(* Logix 5000 project; controller NSH_PLC1 vendor 1 type 14 code 167 rev 32.11; software revision 32.02; part 5 of 12 *)
(* tags used below, declared in another part *)
   H10 : Motor;   // Auger
   H14A : Motor;   // Shr. Roll
   H14B : Motor;   // Shr. Roll
   H15A : Motor;   // Aspirator
   H15B : Motor;   // Aspirator
   H20A : Motor;   // Shr. Roll
   H20B : Motor;   // Shr. Roll
   H20C : Motor;   // Vib.
   H21A : Motor;   // Aspirator
   H21B : Motor;   // Aspirator
   H25 : Motor;   // Ele.
   H26 : Motor;   // Auger
   H27 : Motor;   // Auger
   H28A : Motor;   // HC Vib.
   H28B : Motor;   // Hard Crkr.
   H28C : Motor;   // S.Roll
   H28D : Motor;   // Shr.Roll.
   H29A : Motor;   // Aspirator
   H29B : Motor;   // Aspirator
   H30 : Motor;   // Auger
   H31 : Motor;   // Roll Fdr.
   H32A : Motor;   // HS Cracker
   H32B : Motor;   // Hard Crkr.
   H32C : Motor;   // Shr.Roll.
   H32D : Motor;   // Shr.Roll.
   H33A : Motor;   // Aspirator
   H33B : Motor;   // Aspirator
   H34A : Motor;   // HC Vib.
   H34B : Motor;   // Hard Crkr.
   H34C : Motor;   // S.Roll
   H34D : Motor;   // Shr.Roll.
   H35A : Motor;   // Aspirator
   H35B : Motor;   // Aspirator
   H36 : Motor;   // BMM
   H37A : Motor;   // Aspirator
   H37B : Motor;   // Aspirator
   H38A : Motor;   // Aspirator
   H38B : Motor;   // Aspirator
   H39 : Motor;   // Ele.
   H40 : Motor;   // Auger
   H41 : Motor;   // Auger
   H42A : Motor;   // HC Vib.
   H42B : Motor;   // Hard Crkr.
   H42C : Motor;   // S.Roll
   H42D : Motor;   // Shr.Roll.
   H44A : Motor;   // HC Vib.
   H44B : Motor;   // Hard Crkr.
   H44C : Motor;   // S.Roll
   H44D : Motor;   // Shr.Roll.
   H45A : Motor;   // Aspirator
   H45B : Motor;   // Aspirator
   H46 : Motor;   // BMM
   H47A : Motor;   // Aspirator
   H47B : Motor;   // Aspirator
   H48A : Motor;   // Aspirator
   H48B : Motor;   // Aspirator
(* HullerSheller, continued *)

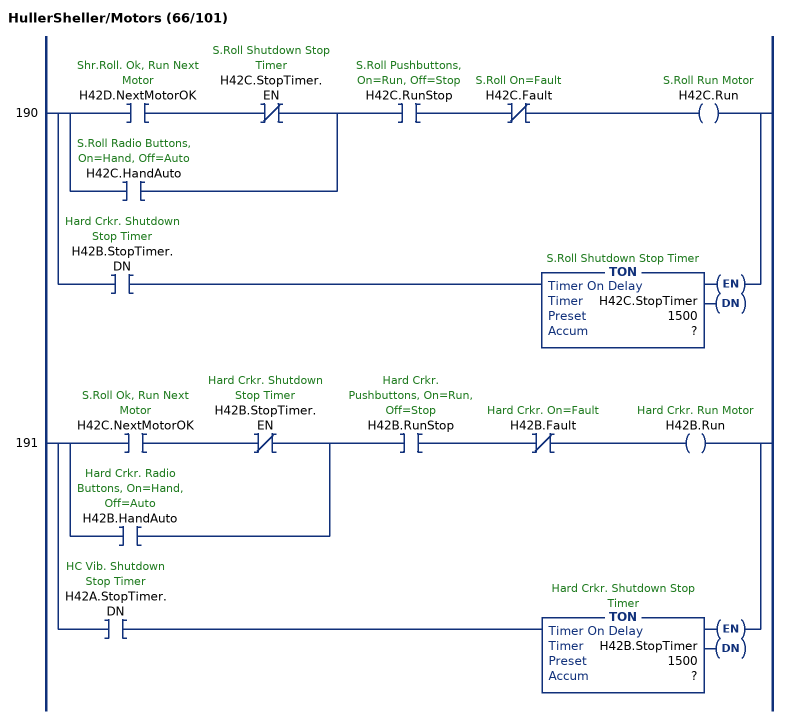
   [picture p90: HullerSheller/Motors rungs 190-191]
   190: [[XIC(H42D.NextMotorOK) XIO(H42C.StopTimer.EN) ,XIC(H42C.HandAuto) ] XIC(H42C.RunStop) XIO(H42C.Fault) OTE(H42C.Run) ,XIC(H42B.StopTimer.DN) TON(H42C.StopTimer,?,?) ];
   191: [[XIC(H42C.NextMotorOK) XIO(H42B.StopTimer.EN) ,XIC(H42B.HandAuto) ] XIC(H42B.RunStop) XIO(H42B.Fault) OTE(H42B.Run) ,XIC(H42A.StopTimer.DN) TON(H42B.StopTimer,?,?) ];
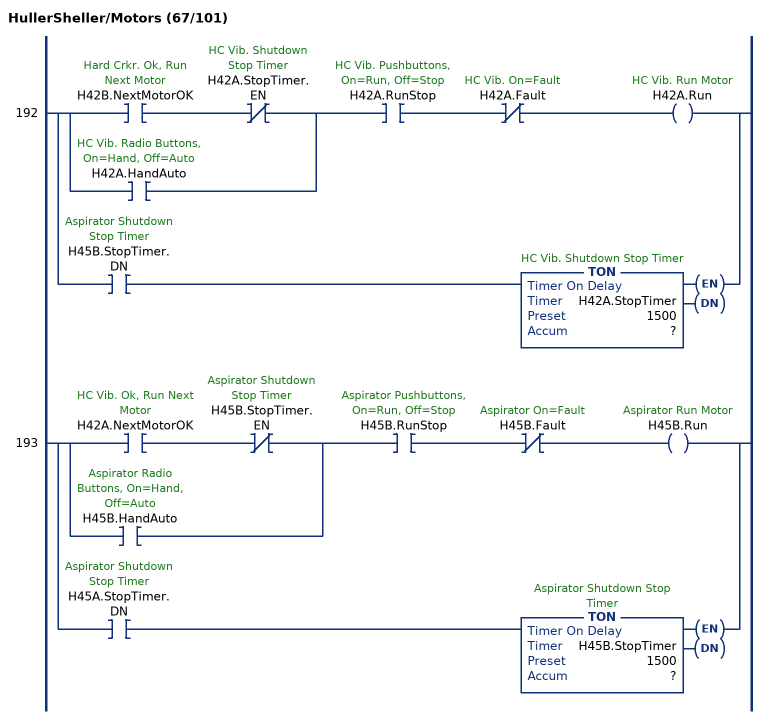
   192: [[XIC(H42B.NextMotorOK) XIO(H42A.StopTimer.EN) ,XIC(H42A.HandAuto) ] XIC(H42A.RunStop) XIO(H42A.Fault) OTE(H42A.Run) ,XIC(H45B.StopTimer.DN) TON(H42A.StopTimer,?,?) ];
   193: [[XIC(H42A.NextMotorOK) XIO(H45B.StopTimer.EN) ,XIC(H45B.HandAuto) ] XIC(H45B.RunStop) XIO(H45B.Fault) OTE(H45B.Run) ,XIC(H45A.StopTimer.DN) TON(H45B.StopTimer,?,?) ];
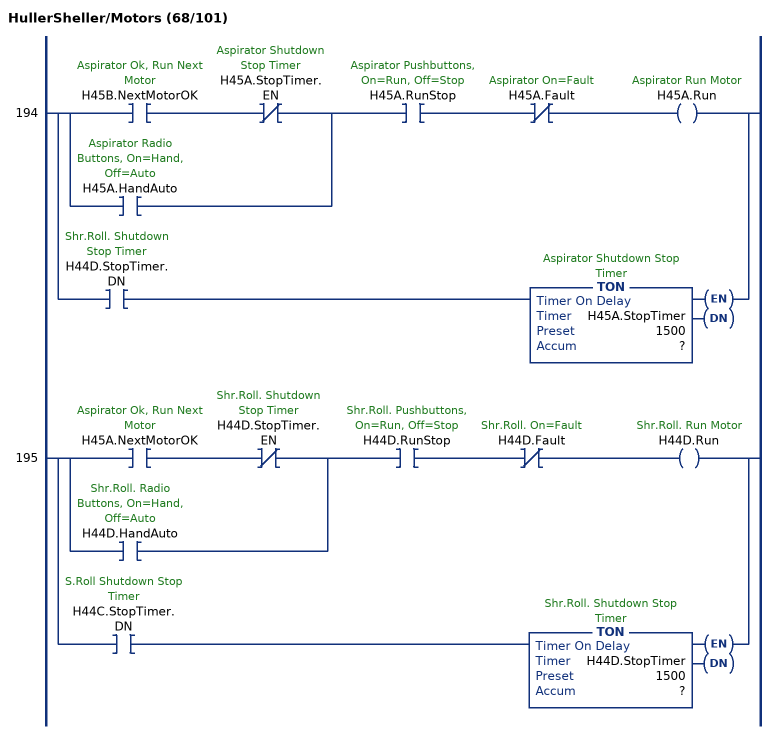
   194: [[XIC(H45B.NextMotorOK) XIO(H45A.StopTimer.EN) ,XIC(H45A.HandAuto) ] XIC(H45A.RunStop) XIO(H45A.Fault) OTE(H45A.Run) ,XIC(H44D.StopTimer.DN) TON(H45A.StopTimer,?,?) ];
   195: [[XIC(H45A.NextMotorOK) XIO(H44D.StopTimer.EN) ,XIC(H44D.HandAuto) ] XIC(H44D.RunStop) XIO(H44D.Fault) OTE(H44D.Run) ,XIC(H44C.StopTimer.DN) TON(H44D.StopTimer,?,?) ];
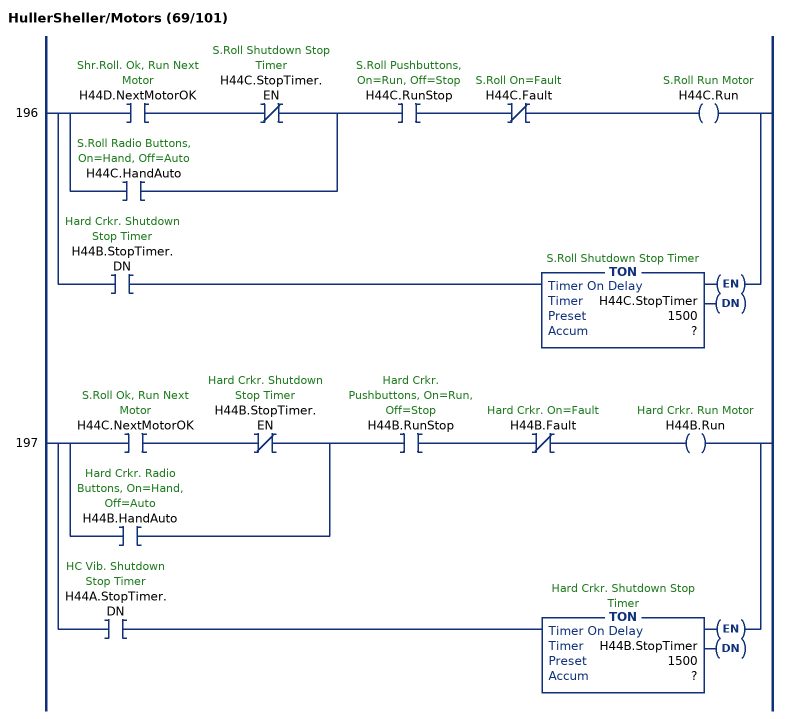
   196: [[XIC(H44D.NextMotorOK) XIO(H44C.StopTimer.EN) ,XIC(H44C.HandAuto) ] XIC(H44C.RunStop) XIO(H44C.Fault) OTE(H44C.Run) ,XIC(H44B.StopTimer.DN) TON(H44C.StopTimer,?,?) ];
   197: [[XIC(H44C.NextMotorOK) XIO(H44B.StopTimer.EN) ,XIC(H44B.HandAuto) ] XIC(H44B.RunStop) XIO(H44B.Fault) OTE(H44B.Run) ,XIC(H44A.StopTimer.DN) TON(H44B.StopTimer,?,?) ];
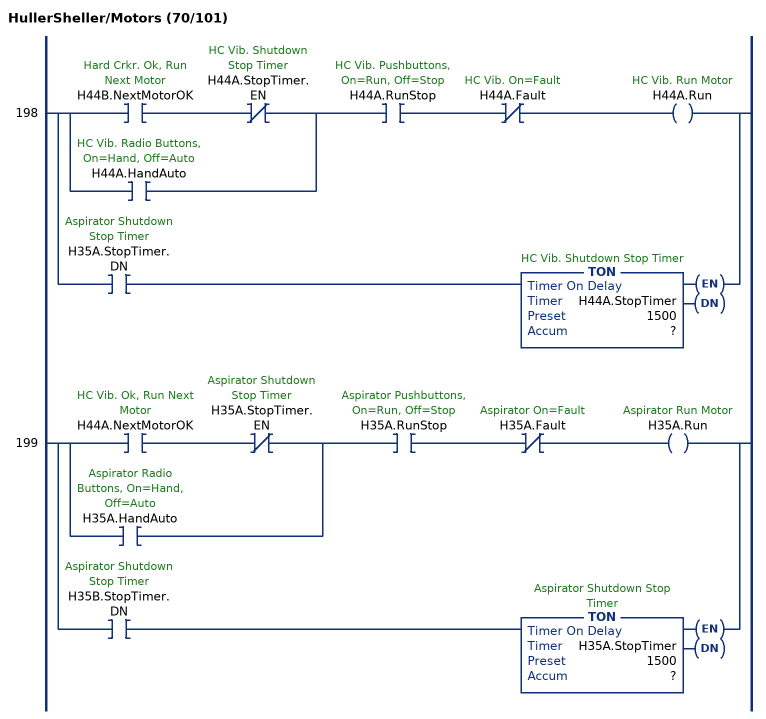
   198: [[XIC(H44B.NextMotorOK) XIO(H44A.StopTimer.EN) ,XIC(H44A.HandAuto) ] XIC(H44A.RunStop) XIO(H44A.Fault) OTE(H44A.Run) ,XIC(H35A.StopTimer.DN) TON(H44A.StopTimer,?,?) ];
   199: [[XIC(H44A.NextMotorOK) XIO(H35A.StopTimer.EN) ,XIC(H35A.HandAuto) ] XIC(H35A.RunStop) XIO(H35A.Fault) OTE(H35A.Run) ,XIC(H35B.StopTimer.DN) TON(H35A.StopTimer,?,?) ];
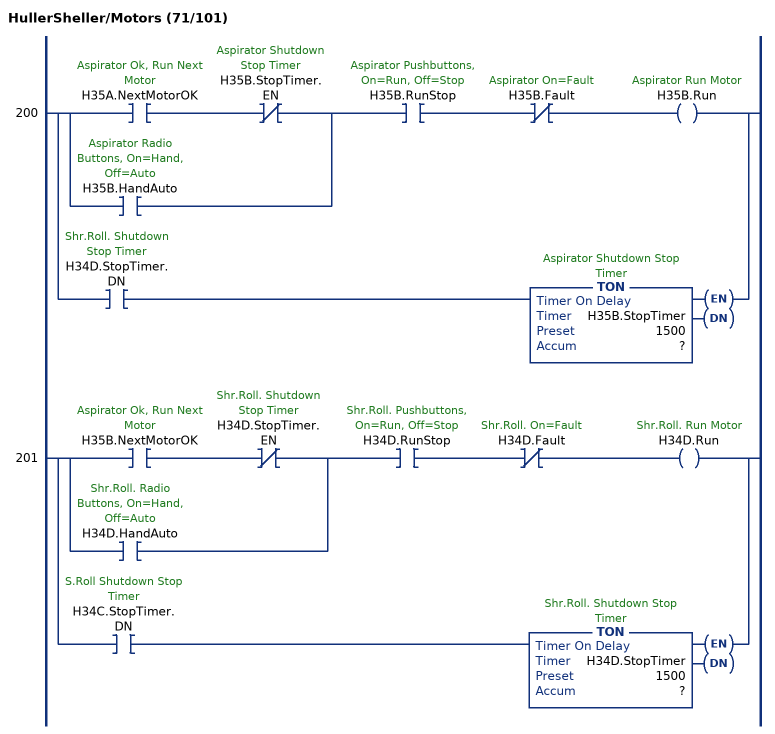
   200: [[XIC(H35A.NextMotorOK) XIO(H35B.StopTimer.EN) ,XIC(H35B.HandAuto) ] XIC(H35B.RunStop) XIO(H35B.Fault) OTE(H35B.Run) ,XIC(H34D.StopTimer.DN) TON(H35B.StopTimer,?,?) ];
   201: [[XIC(H35B.NextMotorOK) XIO(H34D.StopTimer.EN) ,XIC(H34D.HandAuto) ] XIC(H34D.RunStop) XIO(H34D.Fault) OTE(H34D.Run) ,XIC(H34C.StopTimer.DN) TON(H34D.StopTimer,?,?) ];
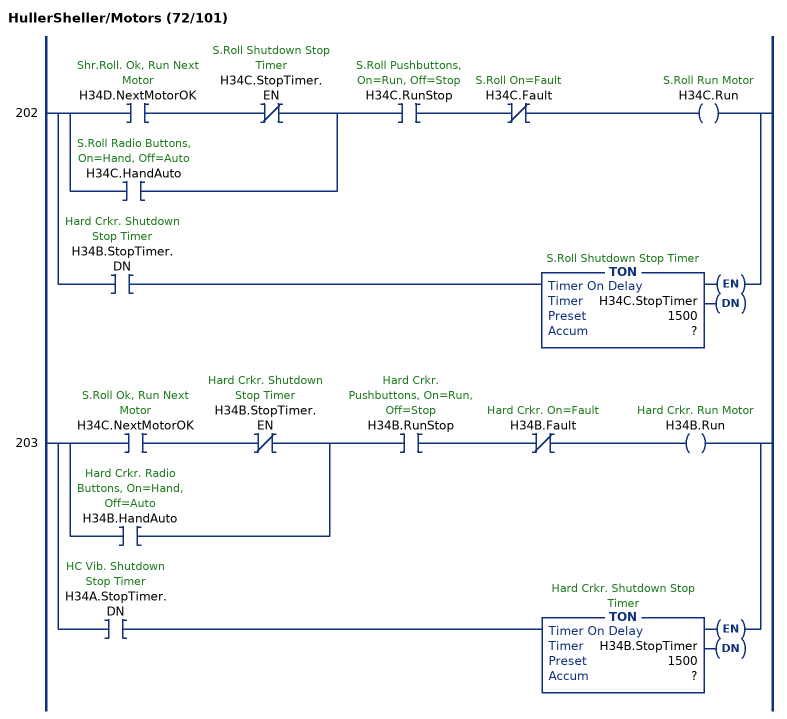
   202: [[XIC(H34D.NextMotorOK) XIO(H34C.StopTimer.EN) ,XIC(H34C.HandAuto) ] XIC(H34C.RunStop) XIO(H34C.Fault) OTE(H34C.Run) ,XIC(H34B.StopTimer.DN) TON(H34C.StopTimer,?,?) ];
   203: [[XIC(H34C.NextMotorOK) XIO(H34B.StopTimer.EN) ,XIC(H34B.HandAuto) ] XIC(H34B.RunStop) XIO(H34B.Fault) OTE(H34B.Run) ,XIC(H34A.StopTimer.DN) TON(H34B.StopTimer,?,?) ];
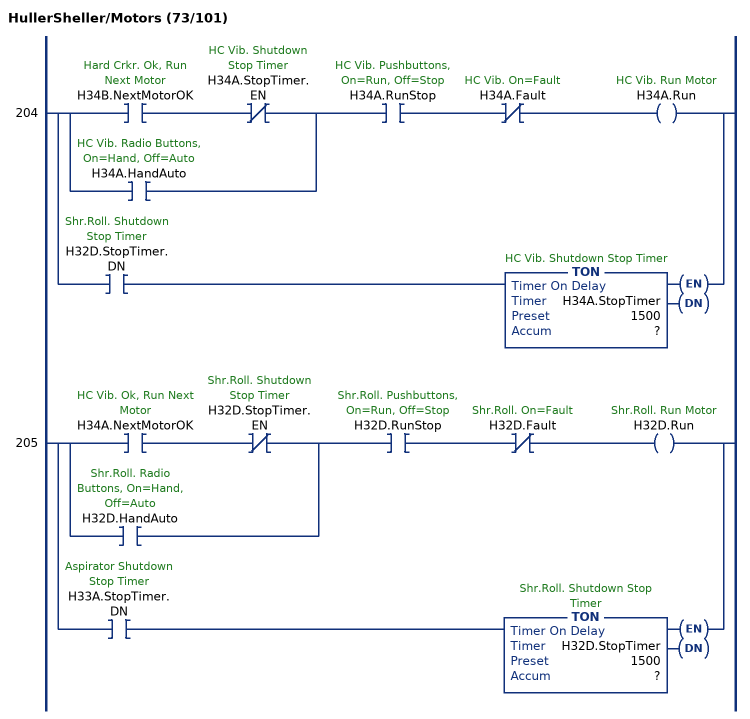
   204: [[XIC(H34B.NextMotorOK) XIO(H34A.StopTimer.EN) ,XIC(H34A.HandAuto) ] XIC(H34A.RunStop) XIO(H34A.Fault) OTE(H34A.Run) ,XIC(H32D.StopTimer.DN) TON(H34A.StopTimer,?,?) ];
   205: [[XIC(H34A.NextMotorOK) XIO(H32D.StopTimer.EN) ,XIC(H32D.HandAuto) ] XIC(H32D.RunStop) XIO(H32D.Fault) OTE(H32D.Run) ,XIC(H33A.StopTimer.DN) TON(H32D.StopTimer,?,?) ];
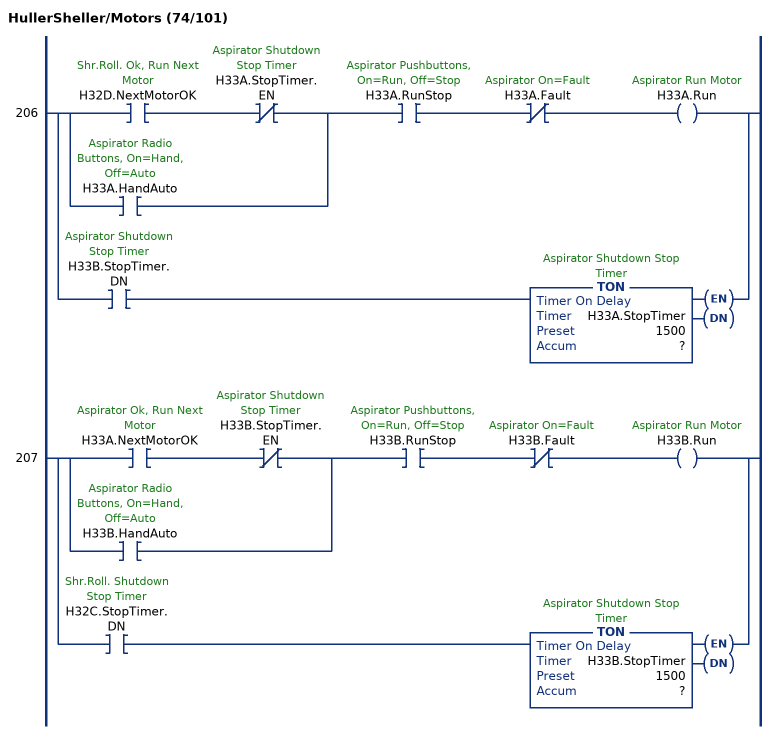
   206: [[XIC(H32D.NextMotorOK) XIO(H33A.StopTimer.EN) ,XIC(H33A.HandAuto) ] XIC(H33A.RunStop) XIO(H33A.Fault) OTE(H33A.Run) ,XIC(H33B.StopTimer.DN) TON(H33A.StopTimer,?,?) ];
   207: [[XIC(H33A.NextMotorOK) XIO(H33B.StopTimer.EN) ,XIC(H33B.HandAuto) ] XIC(H33B.RunStop) XIO(H33B.Fault) OTE(H33B.Run) ,XIC(H32C.StopTimer.DN) TON(H33B.StopTimer,?,?) ];
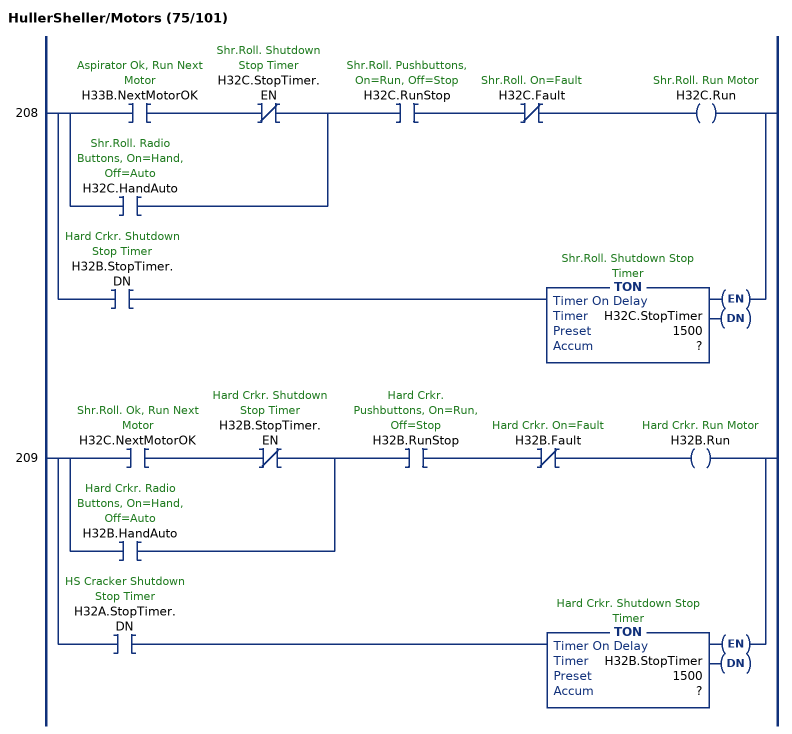
   208: [[XIC(H33B.NextMotorOK) XIO(H32C.StopTimer.EN) ,XIC(H32C.HandAuto) ] XIC(H32C.RunStop) XIO(H32C.Fault) OTE(H32C.Run) ,XIC(H32B.StopTimer.DN) TON(H32C.StopTimer,?,?) ];
   209: [[XIC(H32C.NextMotorOK) XIO(H32B.StopTimer.EN) ,XIC(H32B.HandAuto) ] XIC(H32B.RunStop) XIO(H32B.Fault) OTE(H32B.Run) ,XIC(H32A.StopTimer.DN) TON(H32B.StopTimer,?,?) ];
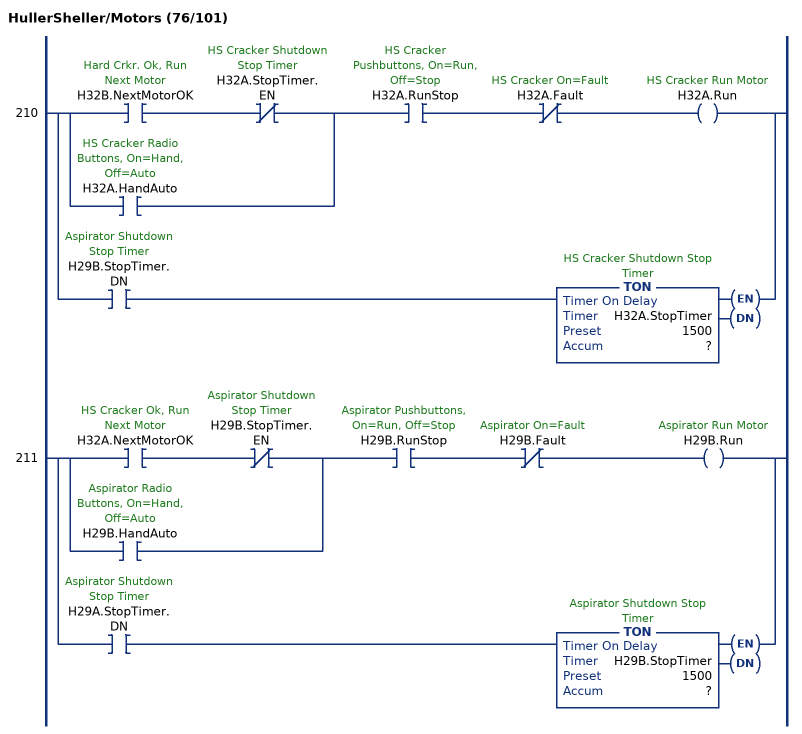
   210: [[XIC(H32B.NextMotorOK) XIO(H32A.StopTimer.EN) ,XIC(H32A.HandAuto) ] XIC(H32A.RunStop) XIO(H32A.Fault) OTE(H32A.Run) ,XIC(H29B.StopTimer.DN) TON(H32A.StopTimer,?,?) ];
   211: [[XIC(H32A.NextMotorOK) XIO(H29B.StopTimer.EN) ,XIC(H29B.HandAuto) ] XIC(H29B.RunStop) XIO(H29B.Fault) OTE(H29B.Run) ,XIC(H29A.StopTimer.DN) TON(H29B.StopTimer,?,?) ];
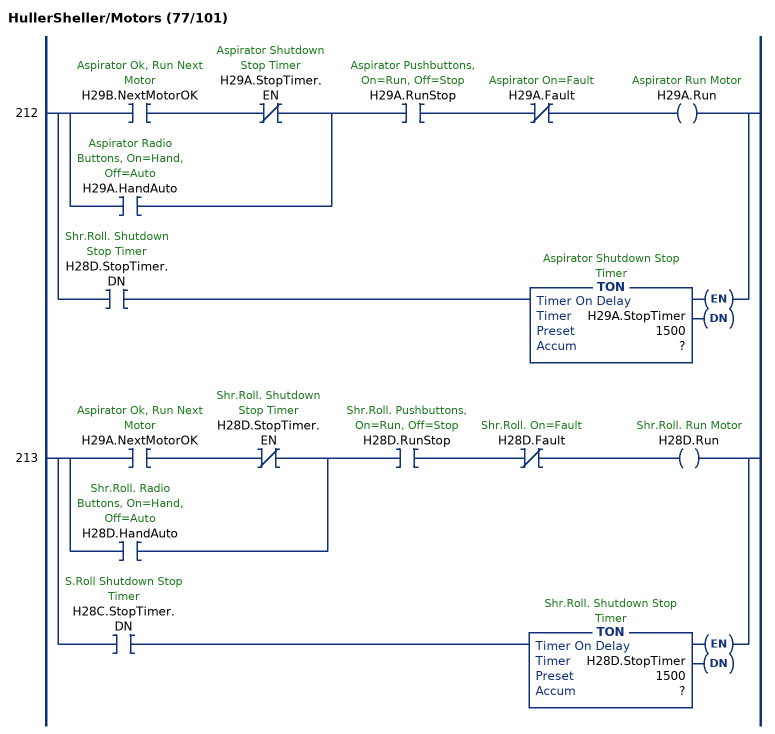
   212: [[XIC(H29B.NextMotorOK) XIO(H29A.StopTimer.EN) ,XIC(H29A.HandAuto) ] XIC(H29A.RunStop) XIO(H29A.Fault) OTE(H29A.Run) ,XIC(H28D.StopTimer.DN) TON(H29A.StopTimer,?,?) ];
   213: [[XIC(H29A.NextMotorOK) XIO(H28D.StopTimer.EN) ,XIC(H28D.HandAuto) ] XIC(H28D.RunStop) XIO(H28D.Fault) OTE(H28D.Run) ,XIC(H28C.StopTimer.DN) TON(H28D.StopTimer,?,?) ];
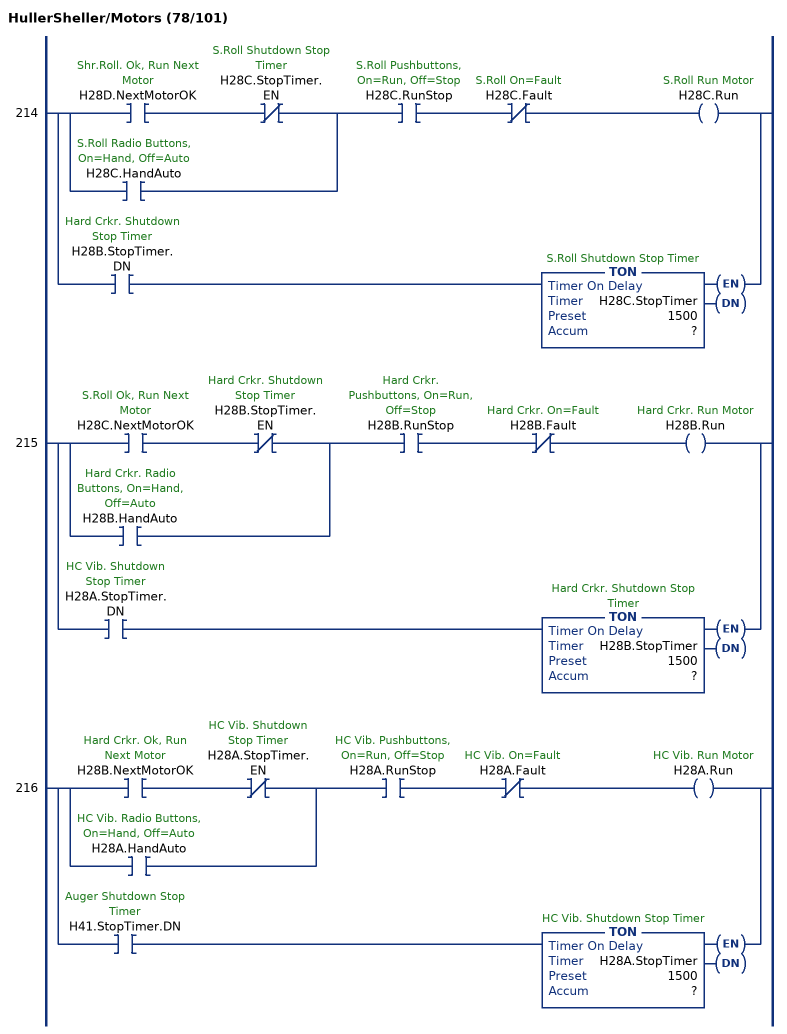
   214: [[XIC(H28D.NextMotorOK) XIO(H28C.StopTimer.EN) ,XIC(H28C.HandAuto) ] XIC(H28C.RunStop) XIO(H28C.Fault) OTE(H28C.Run) ,XIC(H28B.StopTimer.DN) TON(H28C.StopTimer,?,?) ];
   215: [[XIC(H28C.NextMotorOK) XIO(H28B.StopTimer.EN) ,XIC(H28B.HandAuto) ] XIC(H28B.RunStop) XIO(H28B.Fault) OTE(H28B.Run) ,XIC(H28A.StopTimer.DN) TON(H28B.StopTimer,?,?) ];
   216: [[XIC(H28B.NextMotorOK) XIO(H28A.StopTimer.EN) ,XIC(H28A.HandAuto) ] XIC(H28A.RunStop) XIO(H28A.Fault) OTE(H28A.Run) ,XIC(H41.StopTimer.DN) TON(H28A.StopTimer,?,?) ];
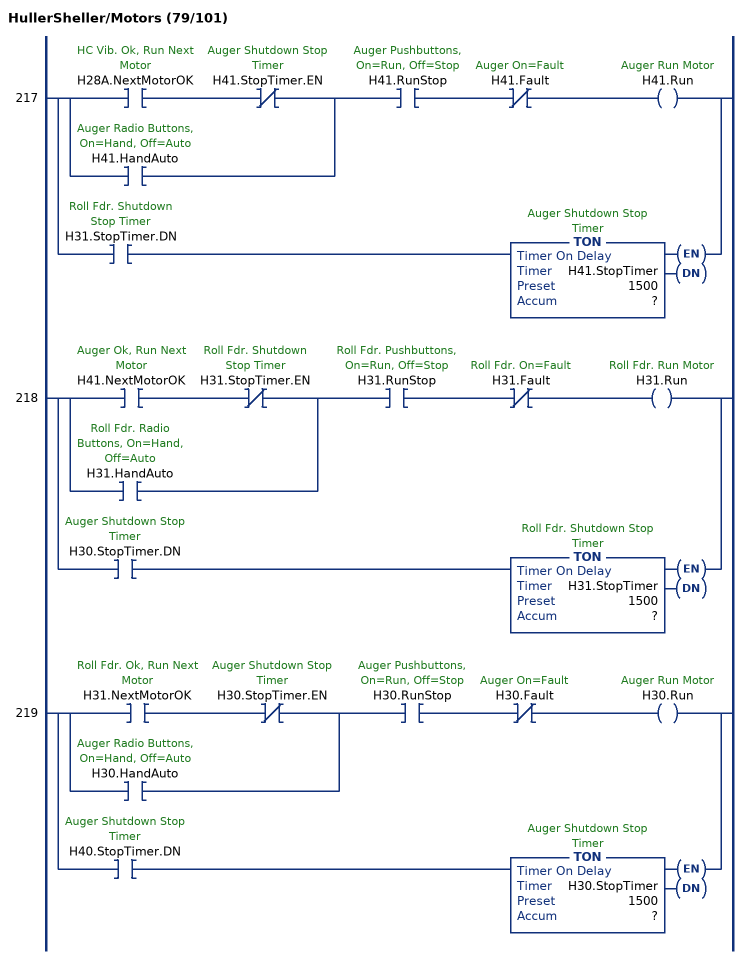
   217: [[XIC(H28A.NextMotorOK) XIO(H41.StopTimer.EN) ,XIC(H41.HandAuto) ] XIC(H41.RunStop) XIO(H41.Fault) OTE(H41.Run) ,XIC(H31.StopTimer.DN) TON(H41.StopTimer,?,?) ];
   218: [[XIC(H41.NextMotorOK) XIO(H31.StopTimer.EN) ,XIC(H31.HandAuto) ] XIC(H31.RunStop) XIO(H31.Fault) OTE(H31.Run) ,XIC(H30.StopTimer.DN) TON(H31.StopTimer,?,?) ];
   219: [[XIC(H31.NextMotorOK) XIO(H30.StopTimer.EN) ,XIC(H30.HandAuto) ] XIC(H30.RunStop) XIO(H30.Fault) OTE(H30.Run) ,XIC(H40.StopTimer.DN) TON(H30.StopTimer,?,?) ];
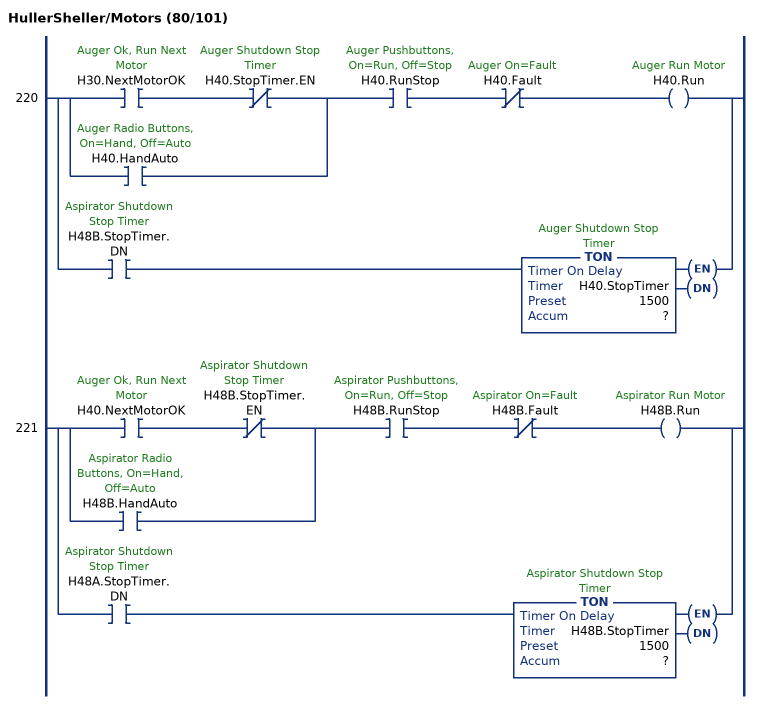
   220: [[XIC(H30.NextMotorOK) XIO(H40.StopTimer.EN) ,XIC(H40.HandAuto) ] XIC(H40.RunStop) XIO(H40.Fault) OTE(H40.Run) ,XIC(H48B.StopTimer.DN) TON(H40.StopTimer,?,?) ];
   221: [[XIC(H40.NextMotorOK) XIO(H48B.StopTimer.EN) ,XIC(H48B.HandAuto) ] XIC(H48B.RunStop) XIO(H48B.Fault) OTE(H48B.Run) ,XIC(H48A.StopTimer.DN) TON(H48B.StopTimer,?,?) ];
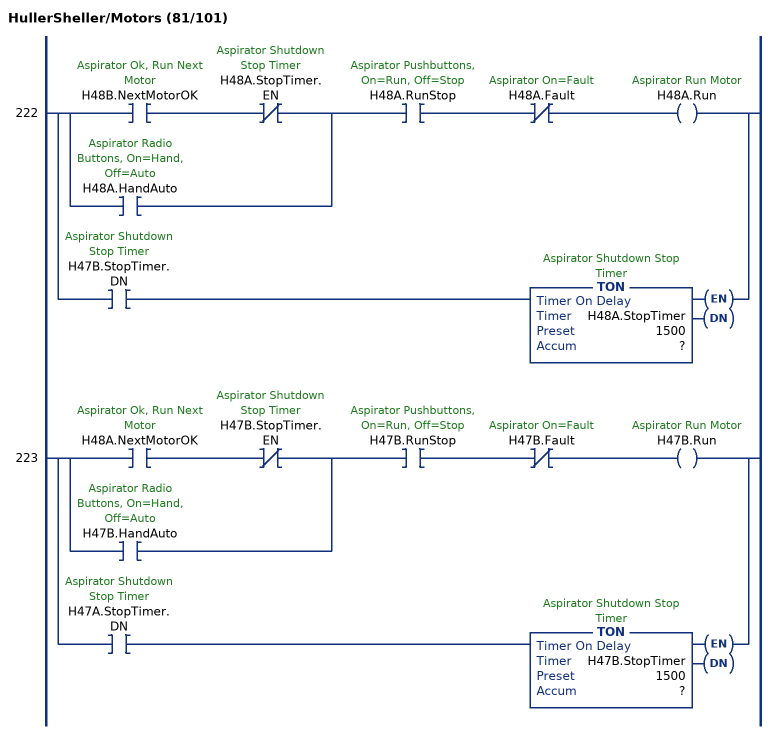
   222: [[XIC(H48B.NextMotorOK) XIO(H48A.StopTimer.EN) ,XIC(H48A.HandAuto) ] XIC(H48A.RunStop) XIO(H48A.Fault) OTE(H48A.Run) ,XIC(H47B.StopTimer.DN) TON(H48A.StopTimer,?,?) ];
   223: [[XIC(H48A.NextMotorOK) XIO(H47B.StopTimer.EN) ,XIC(H47B.HandAuto) ] XIC(H47B.RunStop) XIO(H47B.Fault) OTE(H47B.Run) ,XIC(H47A.StopTimer.DN) TON(H47B.StopTimer,?,?) ];
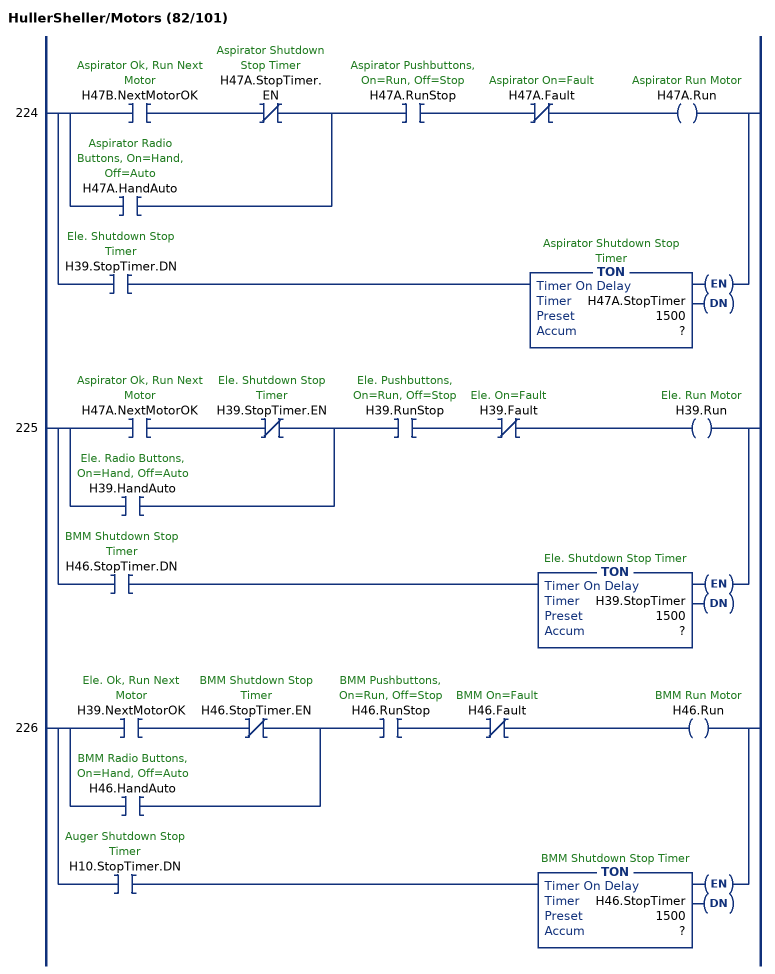
   224: [[XIC(H47B.NextMotorOK) XIO(H47A.StopTimer.EN) ,XIC(H47A.HandAuto) ] XIC(H47A.RunStop) XIO(H47A.Fault) OTE(H47A.Run) ,XIC(H39.StopTimer.DN) TON(H47A.StopTimer,?,?) ];
   225: [[XIC(H47A.NextMotorOK) XIO(H39.StopTimer.EN) ,XIC(H39.HandAuto) ] XIC(H39.RunStop) XIO(H39.Fault) OTE(H39.Run) ,XIC(H46.StopTimer.DN) TON(H39.StopTimer,?,?) ];
   226: [[XIC(H39.NextMotorOK) XIO(H46.StopTimer.EN) ,XIC(H46.HandAuto) ] XIC(H46.RunStop) XIO(H46.Fault) OTE(H46.Run) ,XIC(H10.StopTimer.DN) TON(H46.StopTimer,?,?) ];
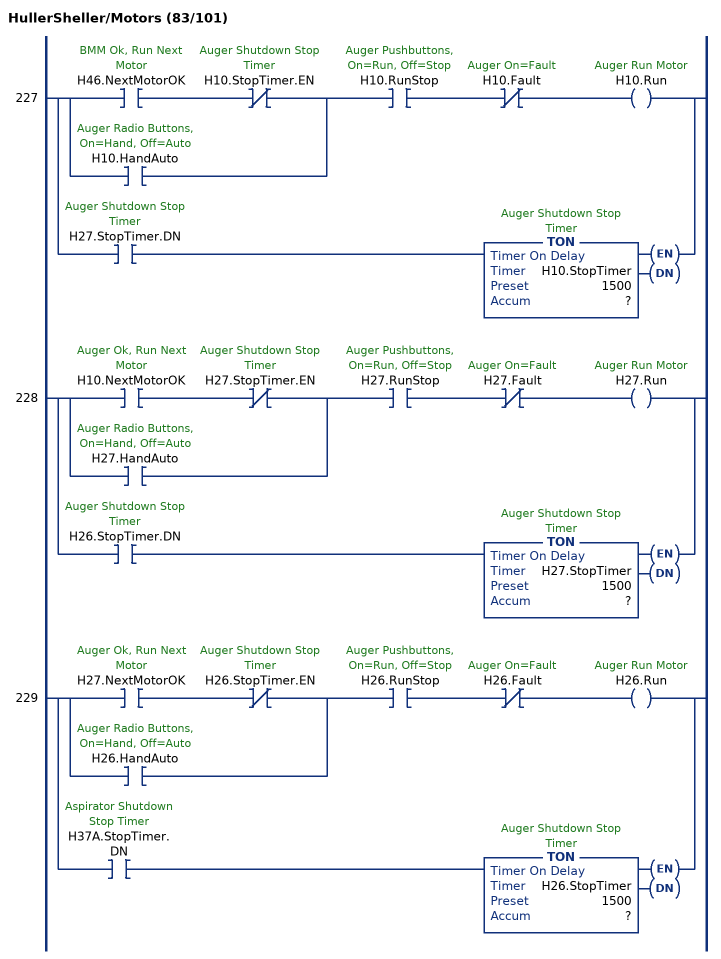
   227: [[XIC(H46.NextMotorOK) XIO(H10.StopTimer.EN) ,XIC(H10.HandAuto) ] XIC(H10.RunStop) XIO(H10.Fault) OTE(H10.Run) ,XIC(H27.StopTimer.DN) TON(H10.StopTimer,?,?) ];
   228: [[XIC(H10.NextMotorOK) XIO(H27.StopTimer.EN) ,XIC(H27.HandAuto) ] XIC(H27.RunStop) XIO(H27.Fault) OTE(H27.Run) ,XIC(H26.StopTimer.DN) TON(H27.StopTimer,?,?) ];
   229: [[XIC(H27.NextMotorOK) XIO(H26.StopTimer.EN) ,XIC(H26.HandAuto) ] XIC(H26.RunStop) XIO(H26.Fault) OTE(H26.Run) ,XIC(H37A.StopTimer.DN) TON(H26.StopTimer,?,?) ];
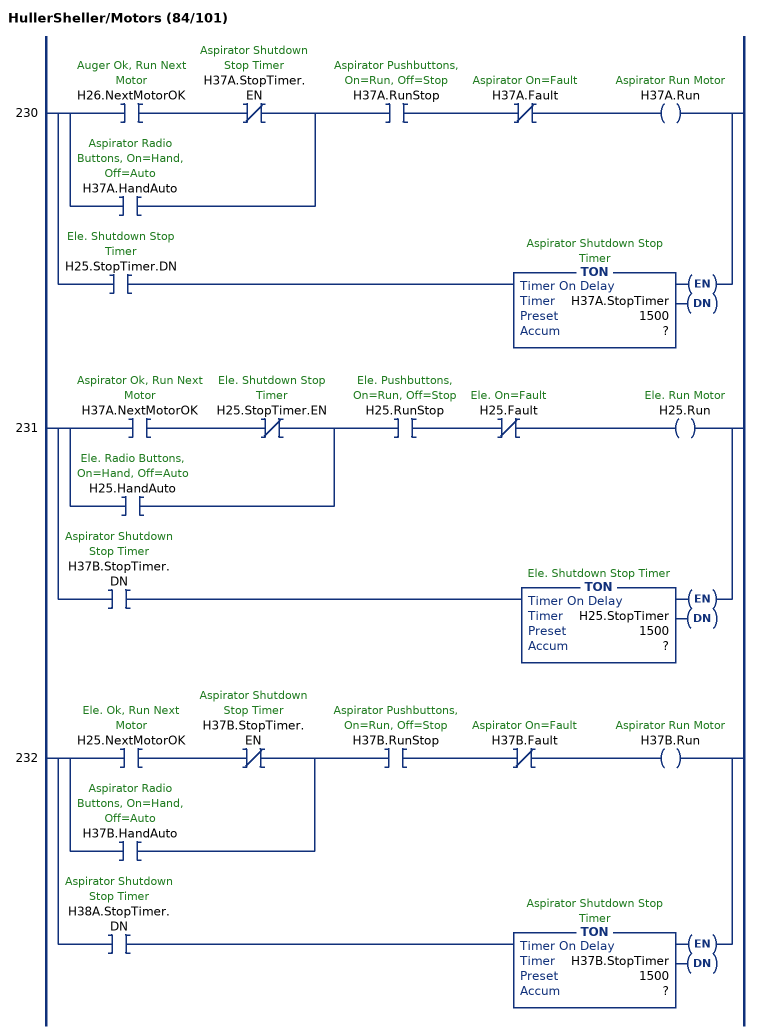
   230: [[XIC(H26.NextMotorOK) XIO(H37A.StopTimer.EN) ,XIC(H37A.HandAuto) ] XIC(H37A.RunStop) XIO(H37A.Fault) OTE(H37A.Run) ,XIC(H25.StopTimer.DN) TON(H37A.StopTimer,?,?) ];
   231: [[XIC(H37A.NextMotorOK) XIO(H25.StopTimer.EN) ,XIC(H25.HandAuto) ] XIC(H25.RunStop) XIO(H25.Fault) OTE(H25.Run) ,XIC(H37B.StopTimer.DN) TON(H25.StopTimer,?,?) ];
   232: [[XIC(H25.NextMotorOK) XIO(H37B.StopTimer.EN) ,XIC(H37B.HandAuto) ] XIC(H37B.RunStop) XIO(H37B.Fault) OTE(H37B.Run) ,XIC(H38A.StopTimer.DN) TON(H37B.StopTimer,?,?) ];
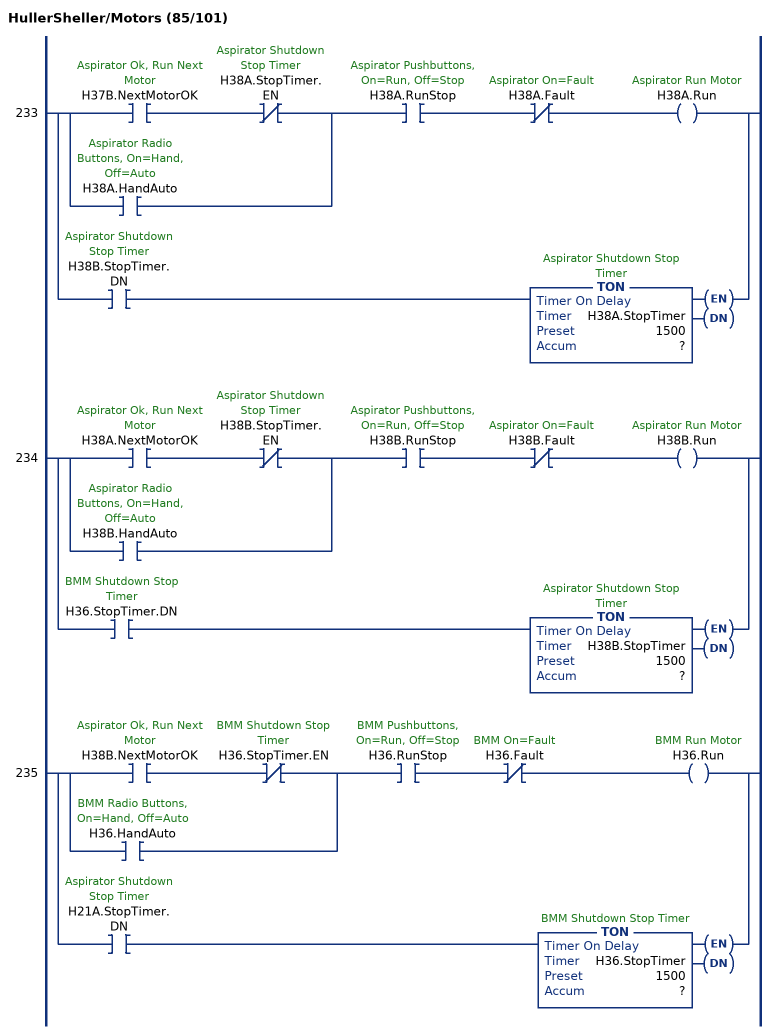
   233: [[XIC(H37B.NextMotorOK) XIO(H38A.StopTimer.EN) ,XIC(H38A.HandAuto) ] XIC(H38A.RunStop) XIO(H38A.Fault) OTE(H38A.Run) ,XIC(H38B.StopTimer.DN) TON(H38A.StopTimer,?,?) ];
   234: [[XIC(H38A.NextMotorOK) XIO(H38B.StopTimer.EN) ,XIC(H38B.HandAuto) ] XIC(H38B.RunStop) XIO(H38B.Fault) OTE(H38B.Run) ,XIC(H36.StopTimer.DN) TON(H38B.StopTimer,?,?) ];
   235: [[XIC(H38B.NextMotorOK) XIO(H36.StopTimer.EN) ,XIC(H36.HandAuto) ] XIC(H36.RunStop) XIO(H36.Fault) OTE(H36.Run) ,XIC(H21A.StopTimer.DN) TON(H36.StopTimer,?,?) ];
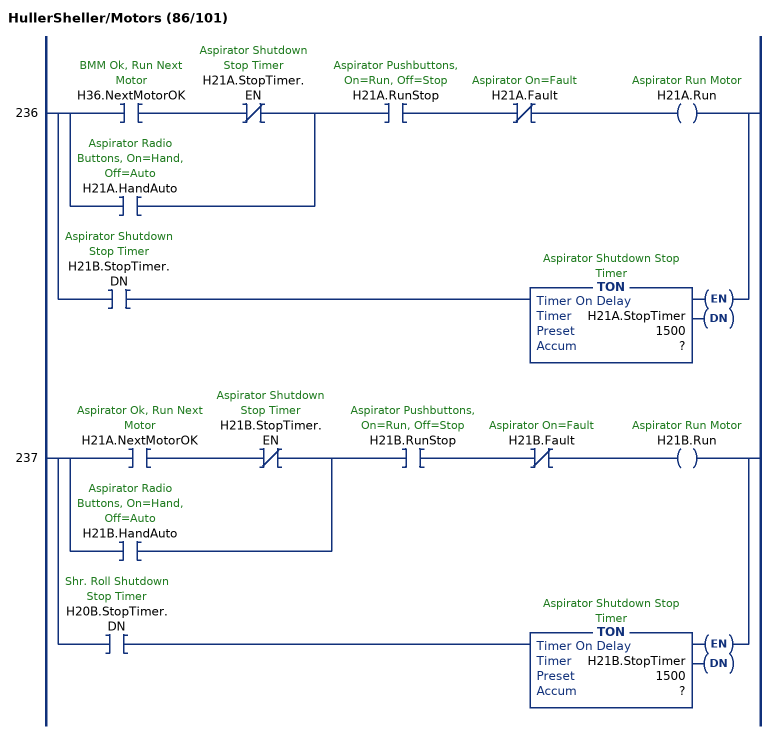
   236: [[XIC(H36.NextMotorOK) XIO(H21A.StopTimer.EN) ,XIC(H21A.HandAuto) ] XIC(H21A.RunStop) XIO(H21A.Fault) OTE(H21A.Run) ,XIC(H21B.StopTimer.DN) TON(H21A.StopTimer,?,?) ];
   237: [[XIC(H21A.NextMotorOK) XIO(H21B.StopTimer.EN) ,XIC(H21B.HandAuto) ] XIC(H21B.RunStop) XIO(H21B.Fault) OTE(H21B.Run) ,XIC(H20B.StopTimer.DN) TON(H21B.StopTimer,?,?) ];
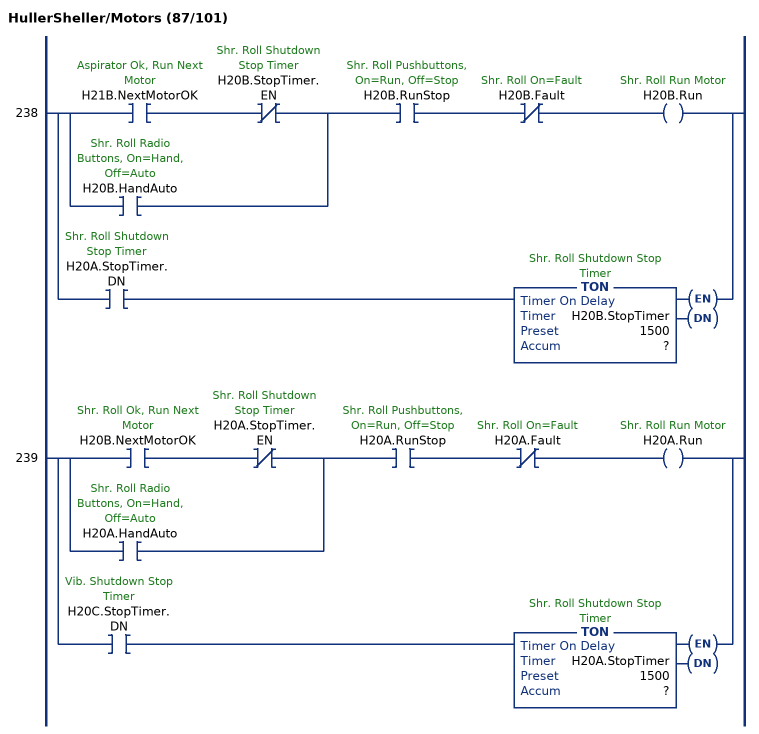
   238: [[XIC(H21B.NextMotorOK) XIO(H20B.StopTimer.EN) ,XIC(H20B.HandAuto) ] XIC(H20B.RunStop) XIO(H20B.Fault) OTE(H20B.Run) ,XIC(H20A.StopTimer.DN) TON(H20B.StopTimer,?,?) ];
   239: [[XIC(H20B.NextMotorOK) XIO(H20A.StopTimer.EN) ,XIC(H20A.HandAuto) ] XIC(H20A.RunStop) XIO(H20A.Fault) OTE(H20A.Run) ,XIC(H20C.StopTimer.DN) TON(H20A.StopTimer,?,?) ];
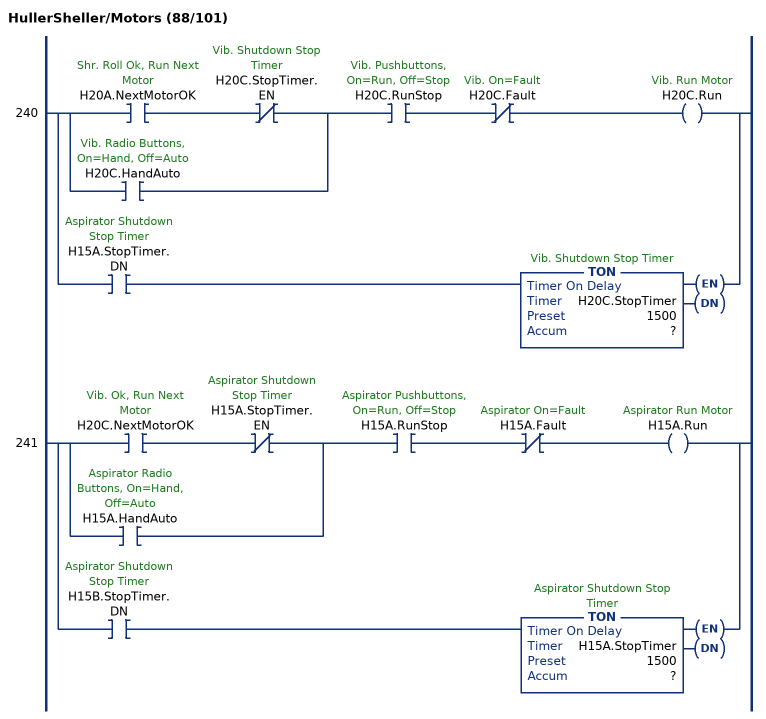
   240: [[XIC(H20A.NextMotorOK) XIO(H20C.StopTimer.EN) ,XIC(H20C.HandAuto) ] XIC(H20C.RunStop) XIO(H20C.Fault) OTE(H20C.Run) ,XIC(H15A.StopTimer.DN) TON(H20C.StopTimer,?,?) ];
   241: [[XIC(H20C.NextMotorOK) XIO(H15A.StopTimer.EN) ,XIC(H15A.HandAuto) ] XIC(H15A.RunStop) XIO(H15A.Fault) OTE(H15A.Run) ,XIC(H15B.StopTimer.DN) TON(H15A.StopTimer,?,?) ];
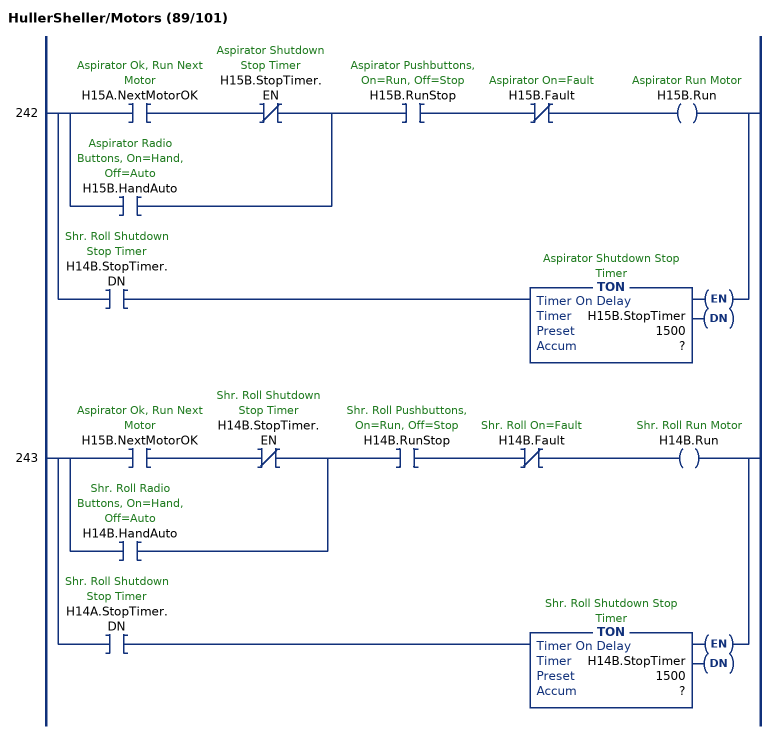
   242: [[XIC(H15A.NextMotorOK) XIO(H15B.StopTimer.EN) ,XIC(H15B.HandAuto) ] XIC(H15B.RunStop) XIO(H15B.Fault) OTE(H15B.Run) ,XIC(H14B.StopTimer.DN) TON(H15B.StopTimer,?,?) ];
   243: [[XIC(H15B.NextMotorOK) XIO(H14B.StopTimer.EN) ,XIC(H14B.HandAuto) ] XIC(H14B.RunStop) XIO(H14B.Fault) OTE(H14B.Run) ,XIC(H14A.StopTimer.DN) TON(H14B.StopTimer,?,?) ];
